// TIA Portal V21 export
FUNCTION_BLOCK "AnalogInput"   // FB903, SCL
{ S7_Optimized_Access := 'TRUE' }
// stored: AutoNumber false, MemoryReserve 100, SetENOAutomatically false
   VAR_INPUT
      simulation { ExternalAccessible := 'False'; ExternalVisible := 'False'; ExternalWritable := 'False'} : Bool;   // Enable simulation input (analog value)
      Reset { ExternalAccessible := 'False'; ExternalVisible := 'False'; ExternalWritable := 'False'} : Bool;
      analogValue { ExternalAccessible := 'False'; ExternalVisible := 'False'; ExternalWritable := 'False'} : Int;   // Input value from sensor (analog signal)
      simulatedAnalogValue { ExternalAccessible := 'False'; ExternalVisible := 'False'; ExternalWritable := 'False'} : Int;   // Simulated analog input value
      Settings { ExternalAccessible := 'False'; ExternalVisible := 'False'; ExternalWritable := 'False'} : "AnalogInputSettings";
   END_VAR
   VAR_OUTPUT
      processValue { ExternalAccessible := 'False'; ExternalVisible := 'False'; ExternalWritable := 'False'} : Real;
      wiringAlarm { ExternalAccessible := 'False'; ExternalVisible := 'False'; ExternalWritable := 'False'} : Bool;
   END_VAR
   VAR
      statAlarm { ExternalAccessible := 'False'; ExternalVisible := 'False'; ExternalWritable := 'False'} : Bool;
      TON_notOK { ExternalAccessible := 'False'; ExternalVisible := 'False'; ExternalWritable := 'False'} : TON_TIME;
      TON_OK { ExternalAccessible := 'False'; ExternalVisible := 'False'; ExternalWritable := 'False'} : TON_TIME;
   END_VAR
   VAR_TEMP
      tempRegValue : Int;
   END_VAR
BEGIN
   REGION Choose input

       #tempRegValue := #analogValue;
       IF #simulation THEN
           #tempRegValue := #simulatedAnalogValue;
       END_IF;

   END_REGION

   REGION Alarm
       #TON_notOK(IN := #Settings.Limits.regMin > #tempRegValue OR #tempRegValue > #Settings.Limits.regMax,
                  PT := #Settings.Limits.regAlarmDelay);

       #TON_OK(IN := #Settings.Limits.regMin < #tempRegValue AND #tempRegValue < #Settings.Limits.regMax AND NOT #TON_notOK.Q,
               PT := #Settings.Limits.regAlarmDelay);

       IF #TON_notOK.Q THEN
           #statAlarm := TRUE;
       ELSIF #TON_OK.Q AND #Reset AND #statAlarm THEN
           #statAlarm := FALSE;
       END_IF;

       #wiringAlarm := #statAlarm;

   END_REGION

   REGION Processing

       IF NOT #Settings.Scaling.Type THEN
           #processValue := #Settings.Scaling.Multiplier * INT_TO_REAL(IN := #tempRegValue);
       ELSE
           #processValue := SCALE_X_REAL(MIN := #Settings.Scaling.valueMin, MAX := #Settings.Scaling.valueMax, VALUE := NORM_X(MIN := #Settings.Scaling.regMin, VALUE := #tempRegValue, MAX := #Settings.Scaling.regMax));

           IF NOT #wiringAlarm THEN
               #processValue := LIMIT_REAL(MN := #Settings.Scaling.valueMin, IN := #processValue, MX := #Settings.Scaling.valueMax);
           END_IF;
       END_IF;

   END_REGION
END_FUNCTION_BLOCK
